Universal Robots URScript: Main Program.script

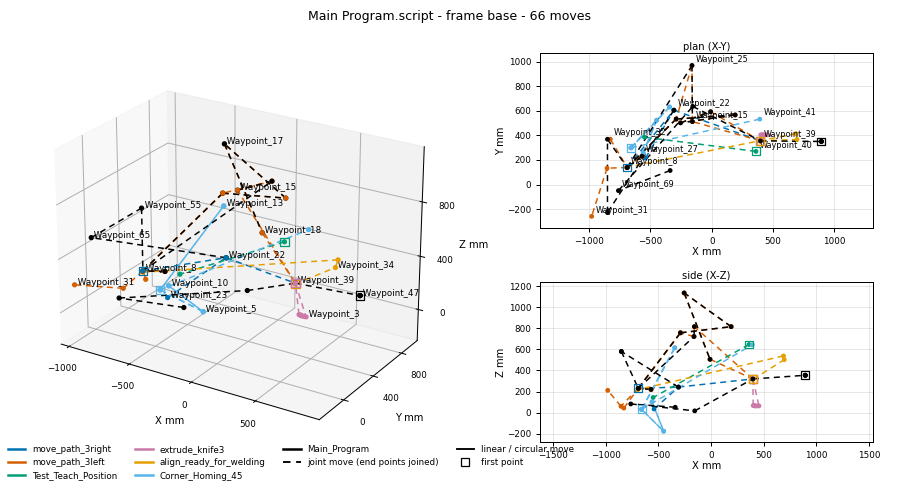
[picture p0: tool path of Main Program.script in frame base, 66 of 133 moves have a stored position in this frame; points joined in program order, loops and branches not executed]
def Main_Program():
  global _hidden_verificationVariable=0
  step_count_c083da12_c088_44e4_86e2_368702bf93a6 = 0.0
  thread Step_Counter_Thread_2b585d60_45ad_46e5_9eb7_fcb77fea0485():
    while (True):
      step_count_c083da12_c088_44e4_86e2_368702bf93a6 = step_count_c083da12_c088_44e4_86e2_368702bf93a6 + 1.0
      sync()
    end
  end
  run Step_Counter_Thread_2b585d60_45ad_46e5_9eb7_fcb77fea0485()
  set_target_payload(10.450000, [0.000000, -0.064000, 0.064000], [0.076889, 0.076889, 0.076889, 0.000000, 0.000000, 0.000000])
  set_tool_communication(False, 115200, 0, 1, 1.5, 3.5)
  set_tool_output_mode(0)
  set_tool_digital_output_mode(0, 1)
  set_tool_digital_output_mode(1, 1)
  set_tool_voltage(0)
  set_safety_mode_transition_hardness(1)
  set_tcp(p[-0.00549,-0.328,0.10639,1.2092,-1.2092,1.2092])
  set_gravity([0.0, 0.0, 9.82])
  set_standard_analog_input_domain(0, 1)
  set_standard_analog_input_domain(1, 1)
  set_tool_analog_input_domain(0, 1)
  set_tool_analog_input_domain(1, 1)
  set_analog_outputdomain(0, 0)
  set_analog_outputdomain(1, 0)
  set_input_actions_to_default()
  global Point_1=p[0.0,0.0,0.0,0.0,0.0,0.0]
  # begin: URCap Installation Node
  #   Source: MachineLogic for Universal Robots, 3.1.7, Vention Inc.
  #   Type: MachineLogic for Universal Robots
  def waitForResponse(expected_response_vention, cname_vention):
  response_vention = socket_read_string(cname_vention,timeout=15)
  while response_vention != expected_response_vention:
  sleep(0.01)
  response_vention = socket_read_string(cname_vention,timeout=15)
  end
  sleep(0.01)
  sync()
  end
  def sendString(string_vention, expected_response_vention, cname_vention):
  socket_send_string(str_cat(string_vention,";"), cname_vention)
  response_vention = socket_read_string(cname_vention,timeout=15)
  if(response_vention == "nAck"):
  popup("nAck received")
  end
  while response_vention != expected_response_vention:
  sleep(0.01)
  response_vention = socket_read_string(cname_vention,timeout=15)
  if(response_vention == "nAck"):
  popup("nAck received")
  end
  end
  sleep(0.01)
  sync()
  end
  def sendStringNAck(string_vention, expected_response_vention, cname_vention):
  socket_send_string(str_cat(string_vention,";"), cname_vention)
  response_vention = socket_read_string(cname_vention,timeout=15)
  if(response_vention == "nAck"):
  popup("nAck received")
  end
  while(response_vention != expected_response_vention and response_vention != "nAck"):
  sleep(0.01)
  response_vention = socket_read_string(cname_vention,timeout=15)
  if(response_vention == "nAck"):
  popup("nAck received",blocking=True)
  end
  end
  sleep(0.01)
  sync()
  end
  def sendStringWithTimeout(string_vention, expected_response_vention, cname_vention):
  socket_send_string(str_cat(string_vention,";"), cname_vention)
  response_vention = socket_read_string(cname_vention,timeout=10)
  if(response_vention == "nAck"):
  popup("nAck received"+string_vention)
  end
  sleep(0.01)
  sync()
  end
  def pollString(string_vention, expected_response_vention, cname_vention):
  socket_send_string(str_cat(string_vention,";"), cname_vention)
  response_vention = socket_read_string(cname_vention,timeout=15)
  if(response_vention == "nAck"):
  popup("nAck received")
  end
  while response_vention != expected_response_vention:
  sleep(1)
  socket_send_string(str_cat(string_vention,";"), cname_vention)
  response_vention = socket_read_string(cname_vention,timeout=15)
  if(response_vention == "nAck"):
  popup("nAck received")
  end
  end
  sleep(0.01)
  sync()
  end
  def sendVariable(var_vention, data_vention, expected_response_vention, cname_vention):
  socket_set_var(var_vention, data_vention, cname_vention)
  response_vention = socket_read_string(cname_vention,timeout=15)
  if(response_vention == "nAck"):
  popup("nAck received")
  end
  while response_vention != expected_response_vention:
  sleep(0.01)
  response_vention = socket_read_string(cname_vention,timeout=15)
  if(response_vention == "nAck"):
  popup("nAck received")
  end
  end
  sleep(0.01)
  sync()
  end
  def intToString(integer_vention,cname_vention):
  stringFix=""
  multiplier_vention123=1
  if integer_vention<0:
  stringFix="-"
  multiplier_vention123=-1
  end
  socket_set_var("GetString",integer_vention*multiplier_vention123,cname_vention)
  string_vention=""
  while string_vention=="":
  sleep(0.01)
  string_vention=socket_read_string(cname_vention,timeout=15)
  end
  sleep(0.01)
  sync()
  string_vention=stringFix+string_vention
  return string_vention
  end
  string_vention=""
  isVentionMovementBusy = False
  isVentionParallelMovementSendingScript = False
  ventionThreadHandle = 1
  isVentionMovementBusyMachineMotion1 = False
  isVentionParallelMovementSendingScriptMachineMotion1 = False
  socket_vention = socket_open("192.168.3.52", 9999, "MachineMotion1")
  if socket_vention==False:
  popup("Check configuration, can't connect to MachineMotion")
  end
  waitForResponse("MachineMotion connection established", "MachineMotion1")
  sendString("isReady", "MachineMotion isReady = true", "MachineMotion1")
  sendStringWithTimeout("setURCapVersion2", "setURCapVersion loaded", "MachineMotion1")
  sendString("SET speed_v2 1000000", "Ack", "MachineMotion1")
  sendString("SET acceleration_v2 100000", "Ack", "MachineMotion1")
  sendString("SET de_axis_1_microsteps_config 8", "Ack", "MachineMotion1")
  sendString("SET de_axis_1_mechanical_gain_config_v2 150000.0", "Ack", "MachineMotion1")
  sendString("SET de_axis_1_direction_config 1", "Ack", "MachineMotion1")
  sendString("SET de_axis_1_type_config Custom Actuator ", "Ack", "MachineMotion1")
  sendString("de_axis_1_config_exec", "Ack", "MachineMotion1")
  # end: URCap Installation Node
  # begin: URCap Installation Node
  #   Source: WireTank Serial, 4.9.0, WireTank, LLC
  #   Type: WireTank Serial
  WTSerialBridge = rpc_factory("xmlrpc","http://127.0.0.1:40511/RPC2")
  # end: URCap Installation Node
  global freedrive_m_var=  False
  global Waypoint_47_p=p[.894110788705, .351078070639, .354441232572, 2.326362155719, 2.052509368646, .057355656444]
  global Waypoint_47_q=[-3.266942326222555, -1.1744836431792756, 1.6532800833331507, 1.0039457517811279, -0.0024531523333948257, -1.5362089315997522]
  global Waypoint_50_p=p[-.568711442653, .230601791901, .220208834751, -1.519093932087, -.535128035721, .573965472012]
  global Waypoint_50_q=[-0.021522347127095998, -1.2794721287539979, 2.4323821703540247, 5.090870934515753, -2.2996109167682093, 1.533644199371338]
  global Waypoint_51_p=p[-.689649894186, .139001107022, .230693120258, -.852023156701, -1.645963115617, 1.645984943001]
  global Waypoint_51_q=[-1.1454814116107386, -1.5427037247321387, 2.8454700152026575, 4.979047852545538, -4.902958456669943, 1.5718834400177002]
  global Waypoint_52_p=p[-.160992057407, .970528182050, .722037363514, -.554955923310, .106486629259, .328544950173]
  global Waypoint_52_q=[-1.2978580633746546, -1.3217003357461472, 2.2583277861224573, 3.7025129038044433, -2.952825371419088, 0.9627944231033325]
  global Waypoint_53_p=p[-.157624488365, .513351401913, .815670293526, -.672704566373, -1.852329693545, -.055423312366]
  global Waypoint_53_q=[-2.7676661650287073, -1.8206430874266566, 2.312763277684347, 1.0122546392628173, -1.0765226523028772, -0.8102834860431116]
  global Waypoint_54_p=p[-.308528116178, .606080777007, .242371251996, -2.133736658076, .349438277129, 2.130953356703]
  global Waypoint_54_q=[-1.9617512861834925, -1.2994225782207032, 2.207935158406393, 0.745708628291748, 1.5955500602722168, 1.41863214969635]
  global Waypoint_65_p=p[-.850299549699, -.229060500451, .580194265918, -.066683564301, -1.566406749139, -.045536147896]
  global Waypoint_65_q=[0.11527767777442932, -1.206728772526123, 2.660132948552267, 3.2525827127644042, -4.69939905801882, -0.18521625200380498]
  global Waypoint_55_p=p[-.850295942693, .369353811615, .580190947871, -.066690142153, -1.566409865149, -.045506050424]
  global Waypoint_55_q=[-0.89636737505068, -1.198587493305542, 2.6061368624316614, 3.3119169908710937, -4.700617257748739, 0.826545238494873]
  global Waypoint_59_p=p[-.689650832419, .138973473550, .230700469426, -.851985360280, -1.645991124348, 1.645990580233]
  global Waypoint_59_q=[-1.1454528013812464, -1.5427289356342335, 2.8454795519458216, 4.979044186859884, -4.902960960065023, 1.5718833208084106]
  global Waypoint_71_p=p[-.289684660393, .534258475721, .757199031184, -.295236718653, -.653013693815, .389426431276]
  global Waypoint_71_q=[-1.3941848913775843, -1.6550847492613734, 2.7336130777942103, 4.156678839320801, -3.798194471989767, 1.7310842275619507]
  global Waypoint_58_p=p[.191120239889, .567518478899, .815512910186, -.135765364935, .396070873472, .208834263225]
  global Waypoint_58_q=[-1.651280705128805, -1.7712346516051234, 2.617981735860006, 3.3066598612019042, -2.656208101903097, 0.8563313484191895]
  global Waypoint_56_p=p[-.254568281661, .502958752129, 1.135400507516, -.261908057482, -.749714619963, 1.349050618455]
  global Waypoint_56_q=[-2.0344861189471644, -1.9012485943236292, 2.469647232686178, 2.2012061315723876, -1.1677187124835413, -0.5094392935382288]
  global Waypoint_57_p=p[-.009221327687, .593713365169, .505808930157, -1.424394189587, -2.344106819810, -.527597949261]
  global Waypoint_57_q=[-2.920837704335348, -1.9932075939574183, 2.3856611887561243, 0.6815890508839111, -0.5688460508929651, -1.1506975332843226]
  global Waypoint_67_p=p[-.339169194335, .114271165560, .051007401747, -.434162127311, 1.872717119498, -1.885153895998]
  global Waypoint_67_q=[-1.410516087208883, -0.9778240484050293, 2.47756010690798, -1.72361483196401, -0.3956816832171839, 1.808600902557373]
  global Waypoint_69_p=p[-.760826542313, -.049762698068, .082649581767, -1.026233921905, -1.612699318499, 1.547123897415]
  global Waypoint_69_q=[-0.22154647508730108, -1.118469015961029, 2.7561236063586634, -1.5568565337783475, -3.851987902318136, 1.559481143951416]
  global Waypoint_70_p=p[-.154414768496, .636923137577, .016979120256, -.302753655748, 1.486961848367, .122240024639]
  global Waypoint_70_q=[-1.1281922499286097, -1.0678585332683106, 2.4290812651263636, -2.7994214497008265, -1.6034835020648401, 1.7401196956634521]
  global Waypoint_49_p=p[.397354147848, .356263001249, .319808682466, 2.316306590727, 2.057646408591, .074101958728]
  global Waypoint_49_q=[-3.4579480330096644, -2.0568953953185023, 2.3266006151782435, -0.2270372670939942, -0.1993797461139124, -0.10534602800478154]
  global Waypoint_48_p=p[.894089819959, .351089510856, .354452935433, 2.326359030986, 2.052526986878, .057346871716]
  global Waypoint_48_q=[-3.266932551060812, -1.1745034915259858, 1.653294865285055, 1.0039614874073486, -0.002454582844869435, -1.5362089315997522]
  global Waypoint_46_p=p[.894107867742, .351078231601, .354456446052, 2.326366960603, 2.052510258679, .057358671808]
  global Waypoint_46_q=[-3.266944233571188, -1.1744955343059083, 1.6532734076129358, 1.003952904338501, -0.002457443867818654, -1.5361955801593226]
  global Waypoint_8_p=p[-.689650873132, .138963273545, .230691387978, -.851994598965, -1.645998530536, 1.646007616333]
  global Waypoint_8_q=[-0.9414032141314905, -1.501500443821289, 2.801856819783346, 4.981602895050802, -4.698942009602682, 1.571649193763733]
  global Waypoint_22_p=p[-.308534453517, .606084664264, .242393158856, 1.369873371142, 1.066881263643, -1.257197506198]
  global Waypoint_22_q=[-1.4685500303851526, -0.9664557737163086, 1.6195090452777308, 0.9282776552387695, 1.6574476957321167, 0.2630845010280609]
  global Waypoint_23_p=p[-.540166575654, .215949141041, .034631452617, -1.505795438113, 1.057579835594, 1.573514753692]
  global Waypoint_23_q=[-0.46167117754091436, -1.1365486842444916, 2.508885685597555, 0.15223841249432368, 1.4952874183654785, 3.819530963897705]
  global Waypoint_24_p=p[-.308525559537, .606096497354, .242373144855, -2.133742737559, .349425192770, 2.130939839044]
  global Waypoint_24_q=[-1.8709262053119105, -1.2877716285041352, 2.192875687276022, 0.7510036665150146, 1.5878156423568726, 1.5091480016708374]
  global Waypoint_39_p=p[.397377312153, .356253310648, .319810281486, 2.316317670744, 2.057592854035, .074120023159]
  global Waypoint_39_q=[-3.4579551855670374, -2.0568958721556605, 2.3265963236438196, -0.22706706941638188, -0.19935590425600225, -0.10534030595888311]
  global Waypoint_37_p=p[.397366630181, .356258644196, .319813668943, 2.316299214281, 2.057614642521, .074125657910]
  global Waypoint_37_q=[-3.4579508940326136, -2.056904455224508, 2.3265963236438196, -0.2270481151393433, -0.19937020937074834, -0.10535222688783819]
  global Waypoint_15_p=p[-.157621040248, .513353603496, .815677694745, -.672699538592, -1.852318447516, -.055422773001]
  global Waypoint_15_q=[-2.770456854497091, -1.8207680187621058, 2.3065691629992884, 1.0170823770710449, -1.0767205397235315, -0.8071182409869593]
  global Waypoint_25_p=p[-.161036555831, .970524399959, .722042384791, -.554954311189, .106465018540, .328580879483]
  global Waypoint_25_q=[-1.3071630636798304, -1.3366777312806626, 2.2083633581744593, 3.7187773424335937, -2.9519384543048304, 0.9132363796234131]
  global Waypoint_72_p=p[-.289685725237, .534256396594, .757196155975, -.295237726329, -.653009715205, .389435972469]
  global Waypoint_72_q=[-1.394179646168844, -1.6550847492613734, 2.7336154619800013, 4.156686468715332, -3.7981911341296595, 1.731092095375061]
  global Waypoint_26_p=p[-.689650873132, .138963273545, .230691387978, -.851994598965, -1.645998530536, 1.646007616333]
  global Waypoint_26_q=[-0.9414032141314905, -1.501500443821289, 2.801856819783346, 4.981602895050802, -4.698942009602682, 1.571649193763733]
  global Waypoint_27_p=p[-.568724745609, .230601805298, .220208295176, -1.519097711196, -.535155391172, .573964121010]
  global Waypoint_27_q=[-0.04883271852602178, -1.2753942471793671, 2.4771457354175013, 5.041022258787908, -2.326899592076437, 1.532160997390747]
  global Waypoint_28_p=p[-.568724745609, .230601805298, .220208295176, -1.519097711196, -.535155391172, .573964121010]
  global Waypoint_28_q=[-0.04883271852602178, -1.2753942471793671, 2.4771457354175013, 5.041022258787908, -2.326899592076437, 1.532160997390747]
  global Waypoint_29_p=p[-.689650873132, .138963273545, .230691387978, -.851994598965, -1.645998530536, 1.646007616333]
  global Waypoint_29_q=[-0.9414032141314905, -1.501500443821289, 2.801856819783346, 4.981602895050802, -4.698942009602682, 1.571649193763733]
  global Waypoint_30_p=p[-.853851193668, .133266829906, .060418082908, -.274178222953, -2.359710051999, .046821166283]
  global Waypoint_30_q=[-0.608560864125387, -1.0122360748103638, 2.787060801182882, 3.7283646303364257, -4.940747324620382, 0.3777344226837158]
  global Waypoint_31_p=p[-.979398188272, -.259625449453, .211289397035, -.673010443572, -1.459355862765, -.640164958946]
  global Waypoint_31_q=[0.36968713998794556, -0.5732358259013672, 2.138303581868307, 3.1253925996967773, -4.70385724702944, -1.2100523153888147]
  global Waypoint_32_p=p[-.826865752305, .369357632284, .043113676955, .574997346548, -1.492225541214, .597128135378]
  global Waypoint_32_q=[-1.0355513731585901, -0.33930082738909917, 2.126244846974508, 2.9386045175739746, -4.711197797452108, 1.7860286235809326]
  global Waypoint_33_p=p[-.689650873132, .138963273545, .230691387978, -.851994598965, -1.645998530536, 1.646007616333]
  global Waypoint_33_q=[-0.9414032141314905, -1.501500443821289, 2.801856819783346, 4.981602895050802, -4.698942009602682, 1.571649193763733]
  global Waypoint_73_p=p[-.289671192632, .534275423553, .757232902417, -.295189983811, -.652980753171, .389398176275]
  global Waypoint_73_q=[-1.39418870607485, -1.65509094814443, 2.7335642019854944, 4.156684561366699, -3.7981610933886927, 1.731088399887085]
  global Waypoint_16_p=p[.191112811238, .567512170908, .815514010937, -.135771161622, .396053809900, .208825693369]
  global Waypoint_16_q=[-1.6536315123187464, -1.762029310266012, 2.6225650946246546, 3.2891055780598144, -2.6549678484546106, 0.8520665764808655]
  global Waypoint_17_p=p[-.254565633623, .502963426820, 1.135401557820, -.261910507478, -.749716086887, 1.349041636154]
  global Waypoint_17_q=[-2.035229508076803, -1.8928028545775355, 2.468372408543722, 2.19391576826062, -1.167032543812887, -0.5091407934771937]
  global Waypoint_18_p=p[-.009208376822, .593717720951, .505810027228, -1.424406033077, -2.344120510145, -.527630245278]
  global Waypoint_18_q=[-2.9172328154193323, -1.9945279560484828, 2.3804522196399134, 0.6930715280720214, -0.5671199003802698, -1.1566088835345667]
  global Waypoint_38_p=p[.397379749540, .356252016937, .319817140705, 2.316310534508, 2.057580214841, .074134378577]
  global Waypoint_38_q=[-3.457958761845724, -2.0569073162474574, 2.3265913168536585, -0.22705944002185063, -0.19935638109316045, -0.10534793535341436]
  global Waypoint_40_p=p[.360688403366, .270119715397, .646144746546, .057805349154, 2.125995180379, 2.134053153683]
  global Waypoint_40_q=[-3.4579489866839808, -2.0569035015501917, 2.3265796343432825, -0.22706706941638188, -0.1993501822101038, -0.10534793535341436]
  global Waypoint_2_p=p[-.548957282596, .386284559177, .143710178207, 1.570800598292, -.000025190822, .000004803470]
  global Waypoint_2_q=[-1.0516188780414026, -1.010990933781006, 2.1562450567828577, -1.143702046280243, -1.0526168982135218, -0.0017235914813440445]
  global Waypoint_20_p=p[.397380247322, .356253634699, .319820846021, 2.316316320871, 2.057594704604, .074118471609]
  global Waypoint_20_q=[-3.457949940358297, -2.056894441644186, 2.32658034959902, -0.2270551484874268, -0.19935208955873662, -0.10533696809877569]
  global Waypoint_3_p=p[.454852104155, .405448828659, .064015413765, 2.316807606413, 2.051392071696, .076664825947]
  global Waypoint_3_q=[-3.274653975163595, -1.5604325172356148, 2.467809502278463, -0.34438879907641606, -0.014281574879781544, -0.6303489843951624]
  global Waypoint_21_p=p[.439068323950, .405460163829, .064006334409, 2.316810979609, 2.051438029044, .076624763552]
  global Waypoint_21_q=[-3.2805374304400843, -1.6257621250548304, 2.5041499773608606, -0.4786943954280396, -0.019728008900777638, -0.46699268022646123]
  global Waypoint_42_p=p[.421302935105, .405445303018, .063010865956, 2.316845912097, 2.051376323407, .076625998808]
  global Waypoint_42_q=[-3.2879136244403284, -1.6787048778929652, 2.5389068762408655, -0.5691380065730591, -0.02675801912416631, -0.35834962526430303]
  global Waypoint_43_p=p[.417011768852, .405435328663, .065002627117, 2.316867113472, 2.051334925313, .076628493429]
  global Waypoint_43_q=[-3.289830032979147, -1.6934038601317347, 2.5445857683764856, -0.579618052845337, -0.028589550648824513, -0.33885270753969365]
  global Waypoint_44_p=p[.413030241071, .405436708516, .067007287168, 2.316842962602, 2.051343797062, .076642826315]
  global Waypoint_44_q=[-3.291628662739889, -1.7069231472411097, 2.5494325796710413, -0.5873385828784485, -0.03035623231996709, -0.3224685827838343]
  global Waypoint_74_p=p[.400006724768, .405435114685, .067002832650, 2.316857393772, 2.051322715522, .076640196251]
  global Waypoint_74_q=[-3.2978647390948694, -1.7389985523619593, 2.5696502367602747, -0.6192590159228821, -0.03645164171327764, -0.27867013612856084]
  global Waypoint_45_p=p[.397380247322, .356253634699, .319820846021, 2.316316320871, 2.057594704604, .074118471609]
  global Waypoint_45_q=[-3.457949940358297, -2.056894441644186, 2.32658034959902, -0.2270551484874268, -0.19935208955873662, -0.10533696809877569]
  global oldhome_p=p[.397683836105, .356251384911, .315246899233, 2.316304177919, 2.057561756051, .074146544723]
  global oldhome_q=[-3.457960907612936, -2.0569125614561976, 2.326589886342184, -0.22707636774096684, -0.19935208955873662, -0.10534269014467412]
  global Waypoint_34_p=p[.695155464390, .367451880816, .502522491683, 2.093108370749, 1.857548644474, .308841595089]
  global Waypoint_34_q=[-3.249415699635641, -1.9387923679747523, 2.3226097265826624, 3.981850786800049, -0.05697328249086553, 1.5286790132522583]
  global Waypoint_35_p=p[.687527620967, .415165960724, .537921070000, 2.127101811831, 1.929915403723, .470130777221]
  global Waypoint_35_q=[-3.249424997960226, -1.9387947521605433, 2.32263428369631, 3.9818588930317382, -6.198007937763826, 1.5286580324172974]
  global Waypoint_36_p=p[-.693756081485, .141369193308, .218584735520, -.851978179689, -1.646001533937, 1.646008371360]
  global Waypoint_36_q=[-1.1533568541156214, -1.4924076360515137, 2.8518698851214808, 4.922323781042852, -4.910887185727255, 1.5719373226165771]
  def calculate_point_to_move_towards(feature, direction, position_distance):
    local posDir=[direction[0], direction[1], direction[2]]
    if (norm(posDir) < 1e-6):
      return get_target_waypoint()
    end
    local direction_vector_normalized=normalize(posDir)
    local displacement_pose=p[direction_vector_normalized[0] * position_distance,direction_vector_normalized[1] * position_distance,direction_vector_normalized[2] * position_distance,0,0,0]
    local wanted_displacement_in_base_frame=pose_sub(pose_trans(feature, displacement_pose), feature)
    return pose_add(get_target_waypoint(), wanted_displacement_in_base_frame)
  end
  global Waypoint_4_p=p[-.658264763546, .299530128456, .030909835036, .426821001551, -1.621505068649, .437070885767]
  global Waypoint_4_q=[-1.350241486226217, -0.9702387017062684, 2.492185179387228, -1.7834822140135707, -0.33723670641054326, 1.8489984273910522]
  global Waypoint_5_p=p[-.448862677341, .524599667441, -.175967040878, 2.473330473302, -1.874382924863, .205319206046]
  global Waypoint_5_q=[-1.1354392210589808, -1.0039964479259034, 2.441021744404928, -2.875528474847311, -1.6043828169452112, 1.7329596281051636]
  global Waypoint_10_p=p[-.559130451394, .259233925829, .102445980692, -.822649281727, -1.486064670292, -.881476138414]
  global Waypoint_10_q=[-0.556256119404928, -1.0744255942157288, 2.9114087263690394, -1.7763501606383265, -4.185837809239523, 1.5288889408111572]
  global Waypoint_11_p=p[-.559130451394, .259233925829, .102445980692, -.822649281727, -1.486064670292, -.881476138414]
  global Waypoint_11_q=[-0.556256119404928, -1.0744255942157288, 2.9114087263690394, -1.7763501606383265, -4.185837809239523, 1.5288889408111572]
  global Waypoint_12_p=p[-.448862677341, .524599667441, -.175967040878, 2.473330473302, -1.874382924863, .205319206046]
  global Waypoint_12_q=[-1.1354392210589808, -1.0039964479259034, 2.441021744404928, -2.875528474847311, -1.6043828169452112, 1.7329596281051636]
  global Waypoint_13_p=p[-.343952006273, .632142227752, .615174722549, -.025948978133, -.008794819136, -.567469912202]
  global Waypoint_13_q=[-1.350241486226217, -0.9702451390079041, 2.492171827946798, -3.0669099293150843, 1.575993537902832, 2.355180025100708]
  global Waypoint_14_p=p[-.343952006273, .632142227752, .615174722549, -.025948978133, -.008794819136, -.567469912202]
  global Waypoint_14_q=[-1.350241486226217, -0.9702451390079041, 2.492171827946798, -3.0669099293150843, 1.575993537902832, 2.355180025100708]
  global Waypoint_41_p=p[.392127936214, .533269017847, .644148583936, .057822570580, 2.125982462550, 2.134033989912]
  global Waypoint_41_q=[-3.4579578081714075, -2.0569120846190394, 2.3265841642962855, -0.22706885755572515, -0.1993349234210413, -0.10534984270204717]
  def move_path_3right():
    $ 118 "move_path_3right" "noBreak"
    $ 119 "'this is the path for Down, Over, then Back Around'"
    # 'this is the path for Down, Over, then Back Around'
    $ 120 "Comment"
    # Comment
    $ 129 "align_ready_for_welding()"
    align_ready_for_welding()
    $ 130 "Comment"
    # Comment
    $ 131 "p1≔pathturn[0]"
    global p1=pathturn[0]
    $ 132 "p2≔pathturn[1]"
    global p2=pathturn[1]
    $ 133 "p4≔pathturn[2]"
    global p4=pathturn[2]
    $ 134 "p5≔pathturn[3]"
    global p5=pathturn[3]
    $ 135 "MoveJ"
    $ 136 "p1" "breakAfter"
    movej(p1, a=1.3962634015954636, v=1.0471975511965976)
    $ 137 "Wait: 8.0"
    sleep(8.0)
    $ 140 "turn_extrusion_on()"
    turn_extrusion_on()
    $ 141 "Set DO[0]=On"
    set_standard_digital_out(0, True)
    $ 142 "MoveL"
    $ 143 "p2" "breakAfter"
    movel(p2, a=0.1, v=0.01)
    # begin: URCap Program Node
    #   Source: WireTank Serial, 4.9.0, WireTank, LLC
    #   Type: WireTank Serial
    $ 144 "Serial Bridge uR0"
    SerialResponse = WTSerialBridge.send_command("/dev/ttyUSB0",1200, 8, "None", "One", "None", 1000, "None", "None", [252,82,48], False)
    # end: URCap Program Node
    $ 145 "Wait: 0.5"
    sleep(0.5)
    $ 146 "Set DO[0]=Off"
    set_standard_digital_out(0, False)
    $ 147 "MoveL"
    $ 148 "p4" "breakAfter"
    movel(p4, a=0.01, v=0.12)
    $ 151 "turn_extrusion_on()"
    turn_extrusion_on()
    $ 152 "Set DO[0]=On"
    set_standard_digital_out(0, True)
    $ 153 "MoveL"
    $ 154 "p5" "breakAfter"
    movel(p5, a=0.1, v=0.01)
    # begin: URCap Program Node
    #   Source: WireTank Serial, 4.9.0, WireTank, LLC
    #   Type: WireTank Serial
    $ 155 "Serial Bridge uR0"
    SerialResponse = WTSerialBridge.send_command("/dev/ttyUSB0",1200, 8, "None", "One", "None", 1000, "None", "None", [252,82,48], False)
    # end: URCap Program Node
    $ 156 "Wait: 2.0"
    sleep(2.0)
    $ 157 "Set DO[0]=Off"
    set_standard_digital_out(0, False)
    $ 158 "Comment"
    # Comment
    $ 159 "pret1≔p[p5[0]+.1,p5[1],p5[2],p5[3],p5[4],p5[5]]"
    global pret1=p[p5[0]+.1,p5[1],p5[2],p5[3],p5[4],p5[5]]
    $ 160 "p_1≔pathturn[4]"
    global p_1=pathturn[4]
    $ 161 "p_2≔pathturn[5]"
    global p_2=pathturn[5]
    $ 162 "p_3≔pathturn[6]"
    global p_3=pathturn[6]
    $ 163 "p_4≔pathturn[7]"
    global p_4=pathturn[7]
    $ 164 "p_5≔pathturn[8]"
    global p_5=pathturn[8]
    $ 165 "p_preheat≔p[p_3[0]+.01,p_3[1],p_3[2],p_3[3],p_3[4],p_3[5]]"
    global p_preheat=p[p_3[0]+.01,p_3[1],p_3[2],p_3[3],p_3[4],p_3[5]]
    $ 166 "p_pre_ret≔p[p_1[0]+.03,p_1[1]+.03,p_1[2],p_1[3],p_1[4],p_1[5]]"
    global p_pre_ret=p[p_1[0]+.03,p_1[1]+.03,p_1[2],p_1[3],p_1[4],p_1[5]]
    $ 167 "p_pre_ret2≔p[p_3[0]+.1,p_3[1],p_3[2],p_3[3],p_3[4],p_3[5]]"
    global p_pre_ret2=p[p_3[0]+.1,p_3[1],p_3[2],p_3[3],p_3[4],p_3[5]]
    $ 168 "MoveJ"
    $ 169 "pret1" "breakAfter"
    movej(pret1, a=1.3962634015954636, v=1.3962634015954636)
    $ 170 "Waypoint_8" "breakAfter"
    movej(get_inverse_kin(Waypoint_8_p, qnear=Waypoint_8_q), a=1.3962634015954636, v=1.0471975511965976)
    $ 172 "Waypoint_22" "breakAfter"
    movej(get_inverse_kin(Waypoint_22_p, qnear=Waypoint_22_q), a=1.3962634015954636, v=1.3962634015954636)
    $ 173 "'preheat'"
    # 'preheat'
    $ 174 "MoveJ"
    $ 175 "p_pre_ret" "breakAfter"
    movej(p_pre_ret, a=1.3962634015954636, v=1.0471975511965976)
    $ 176 "p_pre_ret2" "breakAfter"
    movej(p_pre_ret2, a=1.3962634015954636, v=1.0471975511965976)
    $ 177 "p_preheat" "breakAfter"
    movej(p_preheat, a=1.3962634015954636, v=1.0471975511965976)
    $ 178 "Wait: 8.0"
    sleep(8.0)
    $ 179 "MoveJ"
    $ 180 "p_pre_ret2" "breakAfter"
    movej(p_pre_ret2, a=1.3962634015954636, v=1.0471975511965976)
    $ 181 "p_pre_ret" "breakAfter"
    movej(p_pre_ret, a=1.3962634015954636, v=1.0471975511965976)
    $ 182 "Set"
    set_tcp(p[0.00451,-0.328,0.10639,1.2092,-1.2092,1.2092])
    $ 183 "MoveL"
    $ 184 "p_1" "breakAfter"
    movel(p_1, a=1.2, v=0.05)
    $ 187 "Set DO[0]=On"
    set_standard_digital_out(0, True)
    $ 188 "turn_extrusion_on()"
    turn_extrusion_on()
    $ 189 "MoveL"
    $ 190 "p_2" "breakAfter"
    movel(p_2, a=1.2, v=0.02)
    $ 191 "MoveP"
    $ 192 "CircleMove"
    $ 193 "p_3" "noBreak"
    $ 194 "p_4" "breakAfter"
    movec(p_3, p_4, a=0.01, v=0.001, r=0.0, mode=1)
    $ 195 "MoveL"
    $ 196 "p_5" "breakAfter"
    movel(p_5, a=1.2, v=0.012)
    # begin: URCap Program Node
    #   Source: WireTank Serial, 4.9.0, WireTank, LLC
    #   Type: WireTank Serial
    $ 197 "Serial Bridge uR0"
    SerialResponse = WTSerialBridge.send_command("/dev/ttyUSB0",1200, 8, "None", "One", "None", 1000, "None", "None", [252,82,48], False)
    # end: URCap Program Node
    $ 198 "Wait: 2.0"
    sleep(2.0)
    $ 199 "Set DO[0]=Off"
    set_standard_digital_out(0, False)
    $ 200 "MoveL"
    $ 201 "Waypoint_23" "breakAfter"
    movel(Waypoint_23_p, a=1.2, v=0.25)
    $ 202 "MoveJ"
    $ 203 "Waypoint_24" "breakAfter"
    movej(get_inverse_kin(Waypoint_24_p, qnear=Waypoint_24_q), a=1.3962634015954636, v=1.0471975511965976)
    $ 204 "Waypoint_39" "breakAfter"
    movej(get_inverse_kin(Waypoint_39_p, qnear=Waypoint_39_q), a=1.3962634015954636, v=1.0471975511965976)
    $ 205 "'above waypoint is home'"
    # 'above waypoint is home'
  end
  def move_path_3left():
    $ 206 "move_path_3left" "noBreak"
    $ 207 "'this is the path for Down, Over, then Back Around'"
    # 'this is the path for Down, Over, then Back Around'
    $ 208 "Comment"
    # Comment
    $ 209 "MoveJ"
    $ 210 "Waypoint_37" "breakAfter"
    movej(get_inverse_kin(Waypoint_37_p, qnear=Waypoint_37_q), a=1.3962634015954636, v=1.0471975511965976)
    $ 211 "'above point is home'"
    # 'above point is home'
    $ 212 "Waypoint_15" "breakAfter"
    movej(get_inverse_kin(Waypoint_15_p, qnear=Waypoint_15_q), a=1.3962634015954636, v=1.0471975511965976)
    $ 213 "Waypoint_25" "breakAfter"
    movej(get_inverse_kin(Waypoint_25_p, qnear=Waypoint_25_q), a=1.3962634015954636, v=1.0471975511965976)
    $ 214 "Waypoint_72" "breakAfter"
    movej(get_inverse_kin(Waypoint_72_p, qnear=Waypoint_72_q), a=1.3962634015954636, v=1.0471975511965976)
    $ 215 "Waypoint_26" "breakAfter"
    movej(get_inverse_kin(Waypoint_26_p, qnear=Waypoint_26_q), a=1.3962634015954636, v=1.0471975511965976)
    $ 216 "Waypoint_27" "breakAfter"
    movej(get_inverse_kin(Waypoint_27_p, qnear=Waypoint_27_q), a=1.3962634015954636, v=1.0471975511965976)
    $ 221 "Comment"
    # Comment
    $ 222 "p1≔pathturn[0]"
    global p1=pathturn[0]
    $ 223 "p2≔pathturn[1]"
    global p2=pathturn[1]
    $ 224 "p4≔pathturn[2]"
    global p4=pathturn[2]
    $ 225 "p5≔pathturn[3]"
    global p5=pathturn[3]
    $ 226 "pa1≔p[p1[0]+0.05,p1[1]-0.05,p1[2],p1[3],p1[4],p1[5]]"
    global pa1=p[p1[0]+0.05,p1[1]-0.05,p1[2],p1[3],p1[4],p1[5]]
    $ 227 "MoveJ"
    $ 228 "pa1" "breakAfter"
    movej(pa1, a=1.3962634015954636, v=1.0471975511965976)
    $ 229 "MoveJ"
    $ 230 "p1" "breakAfter"
    movej(p1, a=1.3962634015954636, v=0.2617993877991494)
    $ 231 "Wait: 8.0"
    sleep(8.0)
    $ 234 "turn_extrusion_on()"
    turn_extrusion_on()
    $ 235 "Set DO[0]=On"
    set_standard_digital_out(0, True)
    $ 236 "MoveL"
    $ 237 "p2" "breakAfter"
    movel(p2, a=0.1, v=0.01)
    # begin: URCap Program Node
    #   Source: WireTank Serial, 4.9.0, WireTank, LLC
    #   Type: WireTank Serial
    $ 238 "Serial Bridge uR0"
    SerialResponse = WTSerialBridge.send_command("/dev/ttyUSB0",1200, 8, "None", "One", "None", 1000, "None", "None", [252,82,48], False)
    # end: URCap Program Node
    $ 239 "Wait: 0.5"
    sleep(0.5)
    $ 240 "Set DO[0]=Off"
    set_standard_digital_out(0, False)
    $ 241 "MoveL"
    $ 242 "p4" "breakAfter"
    movel(p4, a=0.01, v=0.12)
    $ 245 "turn_extrusion_on()"
    turn_extrusion_on()
    $ 246 "Set DO[0]=On"
    set_standard_digital_out(0, True)
    $ 247 "MoveL"
    $ 248 "p5" "breakAfter"
    movel(p5, a=0.1, v=0.01)
    # begin: URCap Program Node
    #   Source: WireTank Serial, 4.9.0, WireTank, LLC
    #   Type: WireTank Serial
    $ 249 "Serial Bridge uR0"
    SerialResponse = WTSerialBridge.send_command("/dev/ttyUSB0",1200, 8, "None", "One", "None", 1000, "None", "None", [252,82,48], False)
    # end: URCap Program Node
    $ 250 "Wait: 2.0"
    sleep(2.0)
    $ 251 "Set DO[0]=Off"
    set_standard_digital_out(0, False)
    $ 252 "Comment"
    # Comment
    $ 253 "pret1≔p[p5[0]+.1,p5[1],p5[2],p5[3],p5[4],p5[5]]"
    global pret1=p[p5[0]+.1,p5[1],p5[2],p5[3],p5[4],p5[5]]
    $ 254 "p_1≔pathturn[4]"
    global p_1=pathturn[4]
    $ 255 "p_2≔pathturn[5]"
    global p_2=pathturn[5]
    $ 256 "p_3≔pathturn[6]"
    global p_3=pathturn[6]
    $ 257 "p_4≔pathturn[7]"
    global p_4=pathturn[7]
    $ 258 "p_5≔pathturn[8]"
    global p_5=pathturn[8]
    $ 259 "p_preheat≔p[p_3[0]+.01,p_3[1],p_3[2],p_3[3],p_3[4],p_3[5]]"
    global p_preheat=p[p_3[0]+.01,p_3[1],p_3[2],p_3[3],p_3[4],p_3[5]]
    $ 260 "p_pre_ret≔p[p_1[0]+.03,p_1[1]-.03,p_1[2],p_1[3],p_1[4],p_1[5]]"
    global p_pre_ret=p[p_1[0]+.03,p_1[1]-.03,p_1[2],p_1[3],p_1[4],p_1[5]]
    $ 261 "p_pre_ret2≔p[p_3[0]+.03,p_3[1],p_3[2],p_3[3],p_3[4],p_3[5]]"
    global p_pre_ret2=p[p_3[0]+.03,p_3[1],p_3[2],p_3[3],p_3[4],p_3[5]]
    $ 262 "MoveJ"
    $ 263 "pret1" "breakAfter"
    movej(pret1, a=1.3962634015954636, v=1.3962634015954636)
    $ 264 "Waypoint_28" "breakAfter"
    movej(get_inverse_kin(Waypoint_28_p, qnear=Waypoint_28_q), a=1.3962634015954636, v=1.3962634015954636)
    $ 265 "'now go into the ccw weld position'"
    # 'now go into the ccw weld position'
    $ 266 "Waypoint_29" "breakAfter"
    movej(get_inverse_kin(Waypoint_29_p, qnear=Waypoint_29_q), a=1.3962634015954636, v=1.3962634015954636)
    $ 267 "Comment"
    # Comment
    $ 268 "Waypoint_30" "breakAfter"
    movej(get_inverse_kin(Waypoint_30_p, qnear=Waypoint_30_q), a=1.3962634015954636, v=1.3962634015954636)
    $ 269 "Waypoint_31" "breakAfter"
    movej(get_inverse_kin(Waypoint_31_p, qnear=Waypoint_31_q), a=1.3962634015954636, v=1.3962634015954636)
    $ 278 "MoveL"
    $ 279 "p_pre_ret" "breakAfter"
    movel(p_pre_ret, a=1.2, v=0.25)
    $ 280 "p_pre_ret2" "breakAfter"
    movel(p_pre_ret2, a=1.2, v=0.25)
    $ 281 "p_preheat" "breakAfter"
    movel(p_preheat, a=1.2, v=0.25)
    $ 282 "Wait: 8.0"
    sleep(8.0)
    $ 283 "MoveL"
    $ 284 "p_pre_ret2" "breakAfter"
    movel(p_pre_ret2, a=1.2, v=0.25)
    $ 285 "p_pre_ret" "breakAfter"
    movel(p_pre_ret, a=1.2, v=0.25)
    $ 286 "Set"
    set_tcp(p[0.00451,-0.328,0.10639,1.2092,-1.2092,1.2092])
    $ 287 "MoveL"
    $ 288 "p_1" "breakAfter"
    movel(p_1, a=1.2, v=0.05)
    $ 291 "Set DO[0]=On"
    set_standard_digital_out(0, True)
    $ 292 "turn_extrusion_on()"
    turn_extrusion_on()
    $ 293 "MoveL"
    $ 294 "p_2" "breakAfter"
    movel(p_2, a=1.2, v=0.02)
    $ 295 "MoveP"
    $ 296 "CircleMove"
    $ 297 "p_3" "noBreak"
    $ 298 "p_4" "breakAfter"
    movec(p_3, p_4, a=0.01, v=0.001, r=0.0, mode=1)
    $ 299 "MoveL"
    $ 300 "p_5" "breakAfter"
    movel(p_5, a=1.2, v=0.012)
    # begin: URCap Program Node
    #   Source: WireTank Serial, 4.9.0, WireTank, LLC
    #   Type: WireTank Serial
    $ 301 "Serial Bridge uR0"
    SerialResponse = WTSerialBridge.send_command("/dev/ttyUSB0",1200, 8, "None", "One", "None", 1000, "None", "None", [252,82,48], False)
    # end: URCap Program Node
    $ 302 "Wait: 2.0"
    sleep(2.0)
    $ 303 "Set DO[0]=Off"
    set_standard_digital_out(0, False)
    $ 308 "MoveJ"
    $ 309 "Waypoint_32" "breakAfter"
    movej(get_inverse_kin(Waypoint_32_p, qnear=Waypoint_32_q), a=1.3962634015954636, v=1.0471975511965976)
    $ 310 "Waypoint_33" "breakAfter"
    movej(get_inverse_kin(Waypoint_33_p, qnear=Waypoint_33_q), a=1.3962634015954636, v=1.0471975511965976)
    $ 311 "Waypoint_73" "breakAfter"
    movej(get_inverse_kin(Waypoint_73_p, qnear=Waypoint_73_q), a=1.3962634015954636, v=1.0471975511965976)
    $ 312 "Comment"
    # Comment
    $ 313 "MoveJ"
    $ 314 "Waypoint_16" "breakAfter"
    movej(get_inverse_kin(Waypoint_16_p, qnear=Waypoint_16_q), a=1.3962634015954636, v=1.0471975511965976)
    $ 315 "Waypoint_17" "breakAfter"
    movej(get_inverse_kin(Waypoint_17_p, qnear=Waypoint_17_q), a=1.3962634015954636, v=1.0471975511965976)
    $ 316 "Waypoint_18" "breakAfter"
    movej(get_inverse_kin(Waypoint_18_p, qnear=Waypoint_18_q), a=1.3962634015954636, v=1.0471975511965976)
    $ 317 "Waypoint_38" "breakAfter"
    movej(get_inverse_kin(Waypoint_38_p, qnear=Waypoint_38_q), a=1.3962634015954636, v=1.0471975511965976)
    $ 318 "'above point is home'"
    # 'above point is home'
  end
  def Test_Teach_Position():
    $ 319 "Test_Teach_Position" "noBreak"
    $ 323 "MoveJ"
    $ 324 "Waypoint_40" "breakAfter"
    set_tcp(p[0.0,0.0,0.019,0.0,0.0,0.0])
    movej(get_inverse_kin(Waypoint_40_p, qnear=Waypoint_40_q), a=1.3962634015954636, v=1.0471975511965976)
    $ 325 "'above waypoint is home'"
    # 'above waypoint is home'
    $ 326 "Waypoint_2" "breakAfter"
    set_tcp(p[0.0,0.0,0.019,0.0,0.0,0.0])
    movej(get_inverse_kin(Waypoint_2_p, qnear=Waypoint_2_q), a=1.3962634015954636, v=1.0471975511965976)
    $ 327 "freedrive_m_var≔ False "
    global freedrive_m_var=  False
    $ 328 "freedrive_m_var≔ True "
    global freedrive_m_var=  True
    $ 329 "Popup: Move the robot to the peg center, then click 'Continue'"
    popup("Move the robot to the peg center, then click 'Continue'", "Message", False, False, blocking=True)
    $ 330 "freedrive_m_var≔ False "
    global freedrive_m_var=  False
    $ 331 "Wait: 0.25"
    sleep(0.25)
    $ 332 "sync()"
    sync()
    $ 333 "tcp_pose≔get_actual_joint_positions()"
    global tcp_pose= get_actual_joint_positions ()
  end
  def align_tcp_left():
    $ 334 "align_tcp_left" "noBreak"
    $ 335 "'this program aligns the tcp parallel to the y direction'"
    # 'this program aligns the tcp parallel to the y direction'
    $ 336 "cp≔get_actual_tcp_pose()"
    global cp= get_actual_tcp_pose ()
    $ 337 "aligned_y_pose≔p[cp[0],cp[1],cp[2],1.570796,0,0]"
    global aligned_y_pose=p[cp[0],cp[1],cp[2],1.570796,0,0]
    $ 338 "MoveJ"
    $ 339 "aligned_y_pose" "breakAfter"
    movej(aligned_y_pose, a=1.3962634015954636, v=1.0471975511965976)
  end
  def extrude_knife3():
    $ 340 "extrude_knife3" "noBreak"
    $ 342 "Set"
    set_tcp(p[-0.00549,-0.328,0.10639,1.2092,-1.2092,1.2092])
    $ 343 "MoveJ"
    $ 344 "Waypoint_20" "breakAfter"
    movej(get_inverse_kin(Waypoint_20_p, qnear=Waypoint_20_q), a=1.3962634015954636, v=1.0471975511965976)
    $ 345 "'above waypoint is home'"
    # 'above waypoint is home'
    $ 346 "'move above bucket'"
    # 'move above bucket'
    $ 347 "MoveJ"
    $ 348 "Waypoint_3" "breakAfter"
    movej(get_inverse_kin(Waypoint_3_p, qnear=Waypoint_3_q), a=1.3962634015954636, v=1.0471975511965976)
    $ 349 "'extrude out a foot'"
    # 'extrude out a foot'
    $ 351 "Set DO[0]=On"
    set_standard_digital_out(0, True)
    $ 352 "turn_extrusion_on()"
    turn_extrusion_on()
    $ 353 "Wait: 24.0"
    sleep(24.0)
    # begin: URCap Program Node
    #   Source: WireTank Serial, 4.9.0, WireTank, LLC
    #   Type: WireTank Serial
    $ 354 "Serial Bridge uR0"
    SerialResponse = WTSerialBridge.send_command("/dev/ttyUSB0",1200, 8, "None", "One", "None", 1000, "None", "None", [252,82,48], False)
    # end: URCap Program Node
    $ 355 "Wait: 1.0"
    sleep(1.0)
    $ 356 "Set DO[0]=Off"
    set_standard_digital_out(0, False)
    $ 357 "'slice'"
    # 'slice'
    $ 358 "MoveL"
    $ 359 "Waypoint_21" "breakAfter"
    movel(Waypoint_21_p, a=0.05, v=0.03)
    $ 360 "Waypoint_42" "breakAfter"
    movel(Waypoint_42_p, a=0.05, v=0.03)
    $ 361 "Waypoint_43" "breakAfter"
    movel(Waypoint_43_p, a=0.05, v=0.03)
    $ 362 "Waypoint_44" "breakAfter"
    movel(Waypoint_44_p, a=0.05, v=0.03)
    $ 363 "Waypoint_74" "breakAfter"
    movel(Waypoint_74_p, a=0.05, v=0.03)
    $ 364 "MoveJ"
    $ 365 "Waypoint_45" "breakAfter"
    movej(get_inverse_kin(Waypoint_45_p, qnear=Waypoint_45_q), a=1.3962634015954636, v=1.0471975511965976)
    $ 366 "'above waypoint is home'"
    # 'above waypoint is home'
  end
  def align_tcp_forward():
    $ 368 "align_tcp_forward" "noBreak"
    $ 369 "'this program aligns the tcp parallel to the y direction'"
    # 'this program aligns the tcp parallel to the y direction'
    $ 370 "cp≔get_actual_tcp_pose()"
    global cp= get_actual_tcp_pose ()
    $ 371 "aligned_y_pose≔p[cp[0],cp[1],cp[2],0,-1.570796,0]"
    global aligned_y_pose=p[cp[0],cp[1],cp[2],0,-1.570796,0]
    $ 372 "MoveJ"
    $ 373 "aligned_y_pose" "breakAfter"
    movej(aligned_y_pose, a=1.3962634015954636, v=1.0471975511965976)
  end
  def align_tcp_up():
    $ 374 "align_tcp_up" "noBreak"
    $ 375 "'this program aligns the tcp parallel to the y direction'"
    # 'this program aligns the tcp parallel to the y direction'
    $ 376 "cp≔get_actual_tcp_pose()"
    global cp= get_actual_tcp_pose ()
    $ 377 "aligned_y_pose≔p[cp[0],cp[1],cp[2],0,0,0]"
    global aligned_y_pose=p[cp[0],cp[1],cp[2],0,0,0]
    $ 378 "MoveJ"
    $ 379 "aligned_y_pose" "breakAfter"
    movej(aligned_y_pose, a=1.3962634015954636, v=1.0471975511965976)
  end
  def align_ready_for_welding():
    $ 380 "align_ready_for_welding" "noBreak"
    $ 381 "'this program takes the welder from home to a position alined ready for welding (vertically down)'"
    # 'this program takes the welder from home to a position alined ready for welding (vertically down)'
    $ 382 "MoveJ"
    $ 383 "oldhome" "breakAfter"
    movej(get_inverse_kin(oldhome_p, qnear=oldhome_q), a=1.3962634015954636, v=1.0471975511965976)
    $ 384 "Waypoint_34" "breakAfter"
    movej(get_inverse_kin(Waypoint_34_p, qnear=Waypoint_34_q), a=1.3962634015954636, v=1.0471975511965976)
    $ 385 "Waypoint_35" "breakAfter"
    movej(get_inverse_kin(Waypoint_35_p, qnear=Waypoint_35_q), a=1.3962634015954636, v=1.0471975511965976)
    $ 386 "Waypoint_36" "breakAfter"
    movej(get_inverse_kin(Waypoint_36_p, qnear=Waypoint_36_q), a=1.3962634015954636, v=1.0471975511965976)
  end
  def Corner_Homing_45():
    $ 387 "Corner_Homing_45" "noBreak"
    $ 388 "'Use this program when tool is already positioned close to corner at 45deg'"
    # 'Use this program when tool is already positioned close to corner at 45deg'
    $ 389 "'tool flange will seek all 3 sides. will save those 5 locs in p__'"
    # 'tool flange will seek all 3 sides. will save those 5 locs in p__'
    $ 390 "Set"
    set_tcp(p[0.0,-0.004,0.284,0.0,0.0,0.0])
    $ 391 "'dummy move below for debug'"
    # 'dummy move below for debug'
    $ 396 "Wait: 1.0"
    sleep(1.0)
    $ 397 "tp≔get_actual_tcp_pose()"
    global tp= get_actual_tcp_pose ()
    $ 398 "Script: analyze_touchpoints.script"
    # this file creates the function for analyzing touchpoints
    # define pi
    pi = 3.1415926535

    # this is the main entry point for calculations.
    # it takes in the 5 points, analyzes the shape of the box, and then calculates path points and returns them
    # specifically for Down, Over, then Around (DOtA)
    # specifically for right-sided boxes (vertical weld on right side of edge)
    def main_calculate_right(p11, p12, p21, p22, p3, p13, p23):
        struct1 = analyze_touchpoints_only(p11, p12, p21, p22, p3)
        list1 = analyze_vertical_touchpoints(p11, p12, p13, p21, p22, p23, p3)
        struct2 = calculate_DOtA_points_right(struct1, list1)
        validity = check_validity_right(struct1, struct2)
        return struct2
    end

    # this is the main entry point for calculations.
    # it takes in the 5 points, analyzes the shape of the box, and then calculates path points and returns them
    # specifically for Down, Over, then Around (DOtA)
    # specifically for left-sided boxes (vertical weld on left side of edge)
    def main_calculate_left(p11, p12, p21, p22, p3, p13, p23):
        struct1 = analyze_touchpoints_only(p11, p12, p21, p22, p3)
        list1 = analyze_vertical_touchpoints(p11, p12, p13, p21, p22, p23, p3)
        struct2 = calculate_DOtA_points_left(struct1, list1)
        validity = check_validity_left(struct1, struct2)
        return struct2
    end

    # it takes 5 arguments as points
    # it returns a struct containing: (pointintersect, pointapproach1, pointapproach2, point1, point2, point3, point4, point5, pointreturn1, heading1, heading2, heading3, path2r1, path2r2, path2l1, path2l2)
    # specifically for Around then Up (AtU)
    def analyze_touchpoints(p11, p12, p21, p22, p3):
      # FIND THE INTERSECTION
      # comment get the z
      zcoord=p3[2]

      # get the raw points from the first line
      l1p1x=p11[0]
      l1p1y=p11[1]
      l1p2x=p12[0]
      l1p2y=p12[1]

      # equate the first line in 2d space
      ml1 = (l1p2y-l1p1y) / (l1p2x-l1p1x)

      # b = y - mx
      bl1 = l1p1y - ml1 * l1p1x

      # get the raw points from the second line
      l2p1x=p21[0]
      l2p1y=p21[1]
      l2p2x=p22[0]
      l2p2y=p22[1]

      # equate the second line in 2d space
      ml2 = (l2p2y-l2p1y) / (l2p2x-l2p1x)

      # b = y - mx
      bl2 = l2p1y - ml2 * l2p1x


      # find the intersection of the two lines
      # m1x+b1 = m2x+b2
      # m1x - m2x = b2 - b1
      # x = (b2-b1) / (m1-m2)
      xintersect = (bl2-bl1) / (ml1-ml2)
      yintersect = ml1 * xintersect + bl1

      #FIND THE VECTORS
      #define a vector from the intersection to the second point on the first line
      l1delxfull = l1p2x - xintersect
      l1delyfull = l1p2y - yintersect

      l1delmag = sqrt(l1delxfull*l1delxfull + l1delyfull*l1delyfull)

      l1delxunit = l1delxfull / l1delmag
      l1delyunit = l1delyfull / l1delmag

      #define a vector from the intersection to the second point on the second line
      l2delxfull = l2p2x - xintersect
      l2delyfull = l2p2y - yintersect

      l2delmag = sqrt(l2delxfull*l2delxfull + l2delyfull*l2delyfull)

      l2delxunit = l2delxfull / l2delmag
      l2delyunit = l2delyfull / l2delmag

      # FIND THE FOUR POINTS ON THE LINES
      # find locations 8 inches away from  intersect point
      # CONST
      welddistance = 8
      roundoverdistance = 0.05
      zup = .375
      # inches
      wd = welddistance * 25.4 / 1000
      rod = roundoverdistance * 25.4 / 1000
      zup = zup * 25.4 / 1000

      # now we have the unit vector. extend the weld distance from the intersection
      x = xintersect + l1delxunit * wd
      y = yintersect + l1delyunit * wd
      z = zcoord + zup

      point1 = p[x,y,z,1.570796,0,0] # dummy orientation for now

      x = xintersect + l1delxunit * rod
      y = yintersect + l1delyunit * rod

      point2 = p[x,y,z,1.570796,0,0]

      # now we have the unit vector. extend the weld distance from the intersection
      x = xintersect + l2delxunit * wd
      y = yintersect + l2delyunit * wd

      point5 = p[x,y,z,0,-1.570796,0]

      x = xintersect + l2delxunit * rod
      y = yintersect + l2delyunit * rod

      point4 = p[x,y,z,0,-1.570796,0]

      #DEFINE APPROACH POINTS
      pointintersect = p[xintersect,yintersect,zcoord,0,0,0]
      pointapproach1 = p[xintersect+0.1,yintersect+0.1,z,1.570796,0,0]
      pointapproach2 = p[point1[0], point1[1]+0.1, point1[2], point1[3], point1[4], point1[5]]
      pointreturn1 = p[point5[0]+0.1, point5[1], point5[2], point5[3], point5[4], point5[5]]

      #FIND HEADINGS
      #for each heading, find the angle of the line with respect to the pos x axis. then add/subtract 90 degrees because you want to be perpendicular to that
      headingvector1 = convert_uv_to_heading(l1delxunit, l1delyunit)
      headingvector2 = convert_uv_to_heading(l2delxunit, l2delyunit)
      # find halfway heading
      heading2 = (headingvector1 + headingvector2)/2
      # find headings that the robot should face while traveling, perpendicular to the vectors of the sides of the box
      heading1 = headingvector1 + pi/2
      heading3 = headingvector2 - pi/2

      #FIND POINT 3
      #see if we have to / can find point 3
      findpoint3 = True
      if roundoverdistance == 0:
        findpoint3 = False
      end
      if findpoint3:
        # i need to find the point3 such that the arc from p2 to p3 to p4 is tangent to p1-p2 and p4-p5. making this a smooth path will be good
        # the direction of movement is from pointintersect in the direction of heading2
        # how much movement though? this will depend on whether it is actually a 90 degree angle or not.
        # first, find the perpendicular lines through points 2 and 4
        perp2 = find_perpendicular_line(ml1, point2[0], point2[1])
        perp4 = find_perpendicular_line(ml2, point4[0], point4[1])
        # next, find the intersection of those two lines
        perpintersect = find_intersection(perp2[0], perp2[1], perp4[0], perp4[1])
        radiusofcircle = distance_between(perpintersect[0], perpintersect[1], 0, point2[0], point2[1], 0)
        # find a vector the direction of heading2
        uvx = cos(heading2)
        uvy = sin(heading2)
        # compute point3. pass in negative radius because the direction is into the tank but we want to move from the intersection out to the rounded edge.
        point3coords = add_vectordistance_to_point(perpintersect[0], perpintersect[1], z, uvx, uvy, 0, -1 * radiusofcircle)
        point3 = p[point3coords[0], point3coords[1], point3coords[2], 0, 0, 0]
      end

      #APPLY ACTUAL RXRYRZ TO POINTS
      # convert the headings to rxryrz and insert those values into the relevant points
      rxryrz = convert_heading_to_axang(heading1)
      rx = rxryrz[0]
      ry = rxryrz[1]
      rz = rxryrz[2]
      pointapproach1 = p[pointapproach1[0], pointapproach1[1], pointapproach1[2], rx, ry, rz]
      pointapproach2 = p[pointapproach2[0], pointapproach2[1], pointapproach2[2], rx, ry, rz]
      point1 = p[point1[0], point1[1], point1[2], rx, ry, rz]
      point2 = p[point2[0], point2[1], point2[2], rx, ry, rz]
      rxryrz = convert_heading_to_axang(heading2)
      rx = rxryrz[0]
      ry = rxryrz[1]
      rz = rxryrz[2]
      if findpoint3:
        point3 = p[point3[0], point3[1], point3[2], rx, ry, rz]
      else:
        point3 = point2
      end
      rxryrz = convert_heading_to_axang(heading3)
      rx = rxryrz[0]
      ry = rxryrz[1]
      rz = rxryrz[2]
      point4 = p[point4[0], point4[1], point4[2], rx, ry, rz]
      point5 = p[point5[0], point5[1], point5[2], rx, ry, rz]
      pointreturn1 = p[pointreturn1[0], pointreturn1[1], pointreturn1[2], rx, ry, rz]

      #find path2 (the part that goes up)
      four_vertical_points = find_vertical_points(pointintersect, l1delxunit, l1delyunit, l2delxunit, l2delyunit, zup, wd, heading1, heading3)
      path2r1 = four_vertical_points[0]
      path2r2 = four_vertical_points[1]
      path2l1 = four_vertical_points[2]
      path2l2 = four_vertical_points[3]

      #RETURN STRUCT
      ret = struct(pointintersect=pointintersect, pointapproach1=pointapproach1, pointapproach2=pointapproach2, point1=point1, point2=point2, point3=point3, point4=point4, point5=point5, pointreturn1=pointreturn1, heading1=heading1, heading2=heading2, heading3=heading3, path2r1=path2r1, path2r2=path2r2, path2l1=path2l1, path2l2=path2l2)
      return ret
    end

    # it takes 5 arguments as points
    # it returns a struct containing: (pointintersect, heading1, heading2, heading3, l1delxunit, l1delyunit, l2delxunit, l2delyunit)
    def analyze_touchpoints_only(p11, p12, p21, p22, p3):
      # FIND THE INTERSECTION
      # comment get the z
      zcoord=p3[2]

      # get the raw points from the first line
      l1p1x=p11[0]
      l1p1y=p11[1]
      l1p2x=p12[0]
      l1p2y=p12[1]

      # equate the first line in 2d space
      ml1 = (l1p2y-l1p1y) / (l1p2x-l1p1x)

      # b = y - mx
      bl1 = l1p1y - ml1 * l1p1x

      # get the raw points from the second line
      l2p1x=p21[0]
      l2p1y=p21[1]
      l2p2x=p22[0]
      l2p2y=p22[1]

      # equate the second line in 2d space
      ml2 = (l2p2y-l2p1y) / (l2p2x-l2p1x)

      # b = y - mx
      bl2 = l2p1y - ml2 * l2p1x


      # find the intersection of the two lines
      # m1x+b1 = m2x+b2
      # m1x - m2x = b2 - b1
      # x = (b2-b1) / (m1-m2)
      xintersect = (bl2-bl1) / (ml1-ml2)
      yintersect = ml1 * xintersect + bl1

      pointintersect = p[xintersect,yintersect,zcoord,0,0,0]

      #FIND THE VECTORS
      #define a vector from the intersection to the second point on the first line
      l1delxfull = l1p2x - xintersect
      l1delyfull = l1p2y - yintersect

      l1delmag = sqrt(l1delxfull*l1delxfull + l1delyfull*l1delyfull)

      l1delxunit = l1delxfull / l1delmag
      l1delyunit = l1delyfull / l1delmag

      #define a vector from the intersection to the second point on the second line
      l2delxfull = l2p2x - xintersect
      l2delyfull = l2p2y - yintersect

      l2delmag = sqrt(l2delxfull*l2delxfull + l2delyfull*l2delyfull)

      l2delxunit = l2delxfull / l2delmag
      l2delyunit = l2delyfull / l2delmag

      #FIND HEADINGS
      #for each heading, find the angle of the line with respect to the pos x axis. then add/subtract 90 degrees because you want to be perpendicular to that
      headingvector1 = convert_uv_to_heading(l1delxunit, l1delyunit)
      headingvector2 = convert_uv_to_heading(l2delxunit, l2delyunit)
      # find halfway heading
      heading2 = (headingvector1 + headingvector2)/2
      # find headings that the robot should face while traveling, perpendicular to the vectors of the sides of the box
      heading1 = headingvector1 + pi/2
      heading3 = headingvector2 - pi/2

      #RETURN STRUCT
      ret = struct(pointintersect=pointintersect, heading1=heading1, heading2=heading2, heading3=heading3, l1delxunit=l1delxunit, l1delyunit=l1delyunit, l2delxunit=l2delxunit, l2delyunit=l2delyunit)
      return ret
    end

    # given a struct from analyze_touchpoints_only(), calculate the points
    def calculate_DOtA_points_right(struct1, listleans):
        # get the stuff from the struct
        pointintersect = struct1[0]
        heading1 = struct1[1]
        heading2 = struct1[2]
        heading3 = struct1[3]
        l1delxunit = struct1[4]
        l1delyunit = struct1[5]
        l2delxunit = struct1[6]
        l2delyunit = struct1[7]

        # FIND THE POINTS ON THE LINES OF THE FIRST TURN PATH
        # find locations 8 inches away from  intersect point
        # CONST
        welddistance1 = 8 # vertical weld distance
        welddistance2 = 6 # first path second leg
        welddistance3 = 8 # second path second leg
        zup = .375
        # inches
        wd1 = welddistance1 * 25.4 / 1000
        wd2 = welddistance2 * 25.4 / 1000
        wd3 = welddistance3 * 25.4 / 1000
        zup = zup * 25.4 / 1000

        x = pointintersect[0] + l1delxunit * zup
        y = pointintersect[1] + l1delyunit * zup
        z = pointintersect[2] + zup

        #apply actual rxryrz to points
        # convert the headings to rxryrz and insert those values into the relevant points
        rxryrz = convert_heading_to_axang_preheatdown(heading1)
        rx = rxryrz[0]
        ry = rxryrz[1]
        rz = rxryrz[2]

        point1 = p[x + wd1*listleans[0], y + wd1*listleans[1], z + wd1, rx, ry, rz] # add in the listleans factor to follow the face of the box as we move up
        point2 = p[x, y, z, rx, ry, rz]

        # convert the headings to rxryrz and insert those values into the relevant points
        rxryrz = convert_heading_to_axang_ccw(heading1)
        rx = rxryrz[0]
        ry = rxryrz[1]
        rz = rxryrz[2]

        point4 = p[x, y, z, rx, ry, rz]
        x = x + l1delxunit * wd2
        y = y + l1delyunit * wd2
        point5 = p[x, y, z, rx, ry, rz]

        # FIND THE POINTS ON THE LINES OF THE SECOND AROUND PATH
        roundoverdistance = 0.05
        rod = roundoverdistance * 25.4 / 1000

        # now we have the unit vector. extend the weld distance from the intersection
        x = pointintersect[0] + l1delxunit * (zup)
        y = pointintersect[1] + l1delyunit * zup
        # convert the headings to rxryrz and insert those values into the relevant points
        rxryrz = convert_heading_to_axang(heading1)
        rx = rxryrz[0]
        ry = rxryrz[1]
        rz = rxryrz[2]
        point_1 = p[x, y, z, rx, ry, rz]

        x = pointintersect[0] + l1delxunit * rod
        y = pointintersect[1] + l1delyunit * rod
        point_2 = p[x, y, z, rx, ry, rz]

        # now we have the unit vector. extend the weld distance from the intersection
        x = pointintersect[0] + l2delxunit * wd3
        y = pointintersect[1] + l2delyunit * wd3
        # convert the headings to rxryrz and insert those values into the relevant points
        rxryrz = convert_heading_to_axang(heading3)
        rx = rxryrz[0]
        ry = rxryrz[1]
        rz = rxryrz[2]
        point_5 = p[x, y, z, rx, ry, rz]

        x = pointintersect[0] + l2delxunit * rod
        y = pointintersect[1] + l2delyunit * rod
        point_4 = p[x, y, z, rx, ry, rz]

        #FIND POINT 3
        # by calling analyze_touchpoints()
        atret = analyze_touchpoints(point_2, point_1, point_4, point_5, pointintersect)
        point_3 = atret[5]


        struct2 = struct(point1=point1, point2=point2, point4=point4, point5=point5, point_1=point_1, point_2=point_2, point_3=point_3, point_4=point_4, point_5=point_5)
        return struct2
    end

    # given a struct from analyze_touchpoints_only(), calculate the points
    def calculate_DOtA_points_left(struct1, listleans):
        # get the stuff from the struct
        pointintersect = struct1[0]
        heading1 = struct1[1]
        heading2 = struct1[2]
        heading3 = struct1[3]
        l1delxunit = struct1[4]
        l1delyunit = struct1[5]
        l2delxunit = struct1[6]
        l2delyunit = struct1[7]

        # FIND THE POINTS ON THE LINES OF THE FIRST TURN PATH
        # find locations 8 inches away from  intersect point
        # CONST
        welddistance1 = 8 # vertical weld distance
        welddistance2 = 6 # first path second leg
        welddistance3 = 8 # second path second leg
        zup = .375
        # inches
        wd1 = welddistance1 * 25.4 / 1000
        wd2 = welddistance2 * 25.4 / 1000
        wd3 = welddistance3 * 25.4 / 1000
        zup = zup * 25.4 / 1000

        x = pointintersect[0] + l2delxunit * zup
        y = pointintersect[1] + l2delyunit * zup
        z = pointintersect[2] + zup

        #apply actual rxryrz to points
        # convert the headings to rxryrz and insert those values into the relevant points
        rxryrz = convert_heading_to_axang_preheatdown(heading3)
        rx = rxryrz[0]
        ry = rxryrz[1]
        rz = rxryrz[2]

        point1 = p[x + wd1*listleans[0], y + wd1*listleans[1], z + wd1, rx, ry, rz]
        point2 = p[x, y, z, rx, ry, rz]

        # convert the headings to rxryrz and insert those values into the relevant points
        rxryrz = convert_heading_to_axang(heading3)
        rx = rxryrz[0]
        ry = rxryrz[1]
        rz = rxryrz[2]

        point4 = p[x, y, z, rx, ry, rz]
        x = x + l2delxunit * wd2
        y = y + l2delyunit * wd2
        point5 = p[x, y, z, rx, ry, rz]

        # FIND THE POINTS ON THE LINES OF THE SECOND AROUND PATH
        roundoverdistance = 0.05
        rod = roundoverdistance * 25.4 / 1000

        # now we have the unit vector. extend the weld distance from the intersection
        x = pointintersect[0] + l2delxunit * (zup)
        y = pointintersect[1] + l2delyunit * zup
        # convert the headings to rxryrz and insert those values into the relevant points
        rxryrz = convert_heading_to_axang_ccw(heading3)
        rx = rxryrz[0]
        ry = rxryrz[1]
        rz = rxryrz[2]
        point_1 = p[x, y, z, rx, ry, rz]

        x = pointintersect[0] + l2delxunit * rod
        y = pointintersect[1] + l2delyunit * rod
        point_2 = p[x, y, z, rx, ry, rz]

        # now we have the unit vector. extend the weld distance from the intersection
        x = pointintersect[0] + l1delxunit * wd3
        y = pointintersect[1] + l1delyunit * wd3
        # convert the headings to rxryrz and insert those values into the relevant points
        rxryrz = convert_heading_to_axang_ccw(heading1)
        rx = rxryrz[0]
        ry = rxryrz[1]
        rz = rxryrz[2]
        point_5 = p[x, y, z, rx, ry, rz]

        x = pointintersect[0] + l1delxunit * rod
        y = pointintersect[1] + l1delyunit * rod
        point_4 = p[x, y, z, rx, ry, rz]

        #FIND POINT 3
        # by calling analyze_touchpoints()
        atret = analyze_touchpoints(point_2, point_1, point_4, point_5, pointintersect)
        point_3 = atret[5]
        #point 3 will not have the correct rxryrz though because now the gun needs to be face up.
        rxryrz = convert_heading_to_axang_ccw(heading2)
        rx = rxryrz[0]
        ry = rxryrz[1]
        rz = rxryrz[2]
        point_3 = p[point_3[0], point_3[1], point_3[2], rx, ry, rz]

        struct2 = struct(point1=point1, point2=point2, point4=point4, point5=point5, point_1=point_1, point_2=point_2, point_3=point_3, point_4=point_4, point_5=point_5)
        return struct2
    end

    # this function analyzes the vertical points
    # calculates the slope of the edge in question
    # specifically, for each inch up in the z direction, what is the change in x and change in y direction
    # returns a list of [nx, ny]
    def analyze_vertical_touchpoints(p11, p12, p13, p21, p22, p23, p3):
        # first, find the equations of the planes from the 6 points
        plane1 = findplane(p11, p12, p13)
        plane2 = findplane(p21, p22, p23)
        # Find the Direction Vector of the Line: The direction vector d of the line of intersection can be found by taking the cross product of the normal vectors of each plane (a, b, and c)
        nx = plane1[1]*plane2[2] - plane1[2]*plane2[1]
        ny = plane1[2]*plane2[0] - plane1[0]*plane2[2]
        nz = plane1[0]*plane2[1] - plane1[1]*plane2[0]
        # normalize the vector so the z length is 1
        multiplier = 1 / nz
        nx = nx * multiplier
        ny = ny * multiplier
        nz = nz * multiplier # should become equal to 1
        ret = [nx, ny]
        return ret
    end

    # given 3 points, this finds the plane and its equation
    # rereturns ax + by + cz + d = 0 in a list of [a, b, c, d]
    def findplane(p11, p12, p13):
        # extract coordinates
        x1 = p11[0]
        y1 = p11[1]
        z1 = p11[2]
        x2 = p12[0]
        y2 = p12[1]
        z2 = p12[2]
        x3 = p13[0]
        y3 = p13[1]
        z3 = p13[2]
        # create vectors from the points
        v1x = x2-x1
        v1y = y2-y1
        v1z = z2-z1
        v2x = x3-x1
        v2y = y3-y1
        v2z = z3-z1
        #calculate the normal vector using the cross product
        nx = v1y*v2z - v1z*v2y # i component
        ny = v1z*v2x - v1x*v2z # j component
        nz = v1x*v2y - v1y*v2x # k component
        # calculate d in the plane equation
        d = -1 * (nx*x1 + ny*y1 + nz*z1)
        ret = [nx, ny, nz, d]
        return ret
    end

    # given a heading, (ccw from +x axis), find the mx+b slope
    # fails if exactly vertical
    def get_slope_from_heading(heading):
        return tan(heading)
    end



    # this function finds the points (and rxryrz) of the 2 points (start and end) of vertical weld section
    def find_vertical_points(pointintersect, l1delxunit, l1delyunit, l2delxunit, l2delyunit, offset, wd, heading1, heading3):

      # find right side stuff
      # find the point in 3d space that is .375 up and .375 over
      x = pointintersect[0] + l1delxunit * offset
      y = pointintersect[1] + l1delyunit * offset
      z = pointintersect[2] + offset
      # find rxryrz
      rxryrz = convert_heading_to_axang_preheatup(heading1)
      rx = rxryrz[0]
      ry = rxryrz[1]
      rz = rxryrz[2]
      path2r1 = p[x, y, z, rx, ry, rz]
      path2r2 = p[x, y, z + wd, rx, ry, rz]

      # find left side
      # find the point in 3d space that is .375 up and .375 over
      x = pointintersect[0] + l2delxunit * offset
      y = pointintersect[1] + l2delyunit * offset
      z = pointintersect[2] + offset
      # find rxryrz
      rxryrz = convert_heading_to_axang_preheatup(heading3)
      rx = rxryrz[0]
      ry = rxryrz[1]
      rz = rxryrz[2]
      path2l1 = p[x, y, z, rx, ry, rz]
      path2l2 = p[x, y, z + wd, rx, ry, rz]

      ret = struct(path2r1=path2r1, path2r2=path2r2, path2l1=path2l1, path2l2=path2l2)
      return ret
    end

    # this function converts a unit vector to its heading angle ccw from x+ axis
    # takes uvx and uvy
    # returns heading in radians
    def convert_uv_to_heading(uvx, uvy):
      baseang = atan(uvy/uvx)
      if uvx < 0:
        ang = baseang + pi
      elif uvy < 0:
        ang = baseang + pi * 2
      else:
        ang = baseang
      end
      return ang
    end

    # this function finds the equation of a line, perpendicular to a given line, and going through a given point
    # takes 3 arguments: m (the original line's slope), x (point's x coord), y (point's y coord). the b of the original line is not needed
    # returns a list of [m,b] (the slope and intercept of the new line)
    def find_perpendicular_line(origm, x, y):
      m = (1/origm) * -1
      b = y - m*x
      ret = [m, b]
      return ret
    end

    # this function finds the intersection point between two lines in the xy plane
    # takes 4 arguments: m1, b1, m2, b2
    # returns a list of [x,y] (the point of intersection)
    def find_intersection(m1, b1, m2, b2):
      # m1x+b1 = m2x+b2
      # m1x - m2x = b2 - b1
      # x = (b2-b1) / (m1-m2)
      x = (b2-b1) / (m1-m2)
      y = m1 * x + b1
      ret = [x, y]
      return ret
    end

    # this function finds the distance between 2 points in 3d space
    # it takes 6 arguments: x1, y1, z1, x2, y2, z2
    # it returns a distance
    def distance_between(x1, y1, z1, x2, y2, z2):
      distsquared = (x2-x1)*(x2-x1)+(y2-y1)*(y2-y1)+(z2-z1)*(z2-z1)
      dist = sqrt(distsquared)
      return dist
    end

    # this function takes a point, a unit vector, and a distance, and adds the distance to the point in the direction of the unit vector (3d space)
    # it returns a point as a list of coordinates
    def add_vectordistance_to_point(xi, yi, zi, uvx, uvy, uvz, delta):
      xf = xi + uvx * delta
      yf = yi + uvy * delta
      zf = zi + uvz * delta
      ret = [xf, yf, zf]
      return ret
    end

    # this function converts a heading (ccw radians from the positive x axis) into rxryrz to be put into a point p[]
    # this will point the gun in this heading with the bottom side of the gun facing up.
    # the values used in this program were calculated by doing rotation matrix math in the file on WI-CALVINB10 C. Documents. Theory for converting rotations into axis angle representations
    def convert_heading_to_axang(heading):
     axisxraw = -1 * sin(heading)
     axisyraw = cos(heading) + 1
     axiszraw = sin(heading)

     magnitude = sqrt(axisxraw*axisxraw + axisyraw*axisyraw + axiszraw*axiszraw)

     axisxunit = axisxraw / magnitude
     axisyunit = axisyraw / magnitude
     axiszunit = axiszraw / magnitude

     angle = acos( (cos(heading) - 1) / 2 )

     rxout = axisxunit * angle
     ryout = axisyunit * angle
     rzout = axiszunit * angle

     return [rxout, ryout, rzout]
    end

    # this function converts a heading (ccw radians from the positive x axis) into rxryrz to be put into a point p[]
    # this will point the gun in this heading with the preheat side of the gun tip facing up. Used for welding in a vertical path.
    # the values used in this program were calculated by doing rotation matrix math in the file on WI-CALVINB10 C. Documents. Theory for converting rotations into axis angle representations
    def convert_heading_to_axang_preheatup(heading):
     axisxraw = -sin(heading) + 1
     axisyraw = cos(heading)
     axiszraw = cos(heading)

     magnitude = sqrt(axisxraw*axisxraw + axisyraw*axisyraw + axiszraw*axiszraw)

     axisxunit = axisxraw / magnitude
     axisyunit = axisyraw / magnitude
     axiszunit = axiszraw / magnitude

     angle = acos( (-sin(heading) - 1) / 2 )

     rxout = axisxunit * angle
     ryout = axisyunit * angle
     rzout = axiszunit * angle

     return [rxout, ryout, rzout]
    end

    # this function converts a heading (ccw radians from the positive x axis) into rxryrz to be put into a point p[]
    # this will point the gun in this heading with the preheat side of the gun tip facing down. Used for welding in a vertical path downwards.
    # the values used in this program were calculated by doing rotation matrix math in the file on WI-CALVINB10 C. Documents. Theory for converting rotations into axis angle representations
    def convert_heading_to_axang_preheatdown(heading):
     axisxraw = -sin(heading) - 1
     axisyraw = cos(heading)
     axiszraw = -cos(heading)

     magnitude = sqrt(axisxraw*axisxraw + axisyraw*axisyraw + axiszraw*axiszraw)

     axisxunit = axisxraw / magnitude
     axisyunit = axisyraw / magnitude
     axiszunit = axiszraw / magnitude

     angle = acos( (sin(heading) - 1) / 2 )

     rxout = axisxunit * angle
     ryout = axisyunit * angle
     rzout = axiszunit * angle

     return [rxout, ryout, rzout]
    end

    # this function converts a heading (ccw radians from the positive x axis) into rxryrz to be put into a point p[]
    # this will point the gun in this heading with the preheat side of the gun tip facing right. Used for welding counterclockwise around the box.
    # the values used in this program were calculated by doing rotation matrix math in the file on WI-CALVINB10 C. Documents. Theory for converting rotations into axis angle representations
    def convert_heading_to_axang_ccw(heading):
     axisxraw = -sin(heading)
     axisyraw = cos(heading) - 1
     axiszraw = -sin(heading)

     magnitude = sqrt(axisxraw*axisxraw + axisyraw*axisyraw + axiszraw*axiszraw)

     axisxunit = axisxraw / magnitude
     axisyunit = axisyraw / magnitude
     axiszunit = axiszraw / magnitude

     angle = acos( (-cos(heading) - 1) / 2 )

     rxout = axisxunit * angle
     ryout = axisyunit * angle
     rzout = axiszunit * angle

     return [rxout, ryout, rzout]
    end

    # this function is for getting the points along the path of the corner homing 45
    # point0 is the point where they touched
    def get_corner_homing_45_pathpoints(point0):
      p0x = point0[0]
      p0y = point0[1]
      p0z = point0[2]
      p0rx = point0[3]
      p0ry = point0[4]
      p0rz = point0[5]

      #constants
      #distances of how far away from point the touchpoints are
      d0 = 0.10 # how far from the box to retreat and approach
      d1 = 0.03 # first distance from init point
      d2 = 0.15 # second distance from init point
      d3 = 0.125 #vertical distance from first point
      sqrt2 = 0.707106781 # 1/sqrt(2) , the inverse of the sqrt(2)

      ph1 = p[p0x + d0, p0y, p0z + d1, p0rx, p0ry, p0rz] #approach point for turn

      ph2 = p[p0x+d0-d0*0.5-sqrt2*d1, p0y+d0*0.5+sqrt2*d1, p0z+d1, 1.446, -0.8, -0.733]
      ph3 = p[p0x+d0-d0*0.5-sqrt2*d2, p0y+d0*0.5+sqrt2*d2, p0z+d1, 1.446, -0.8, -0.733]
      ph4 = p[p0x+d0-d0*0.5-sqrt2*d1, p0y-d0*0.5-sqrt2*d1, p0z+d1, 0.626, -1.993, -1.813]
      ph5 = p[p0x+d0-d0*0.5-sqrt2*d2, p0y-d0*0.5-sqrt2*d2, p0z+d1, 0.626, -1.993, -1.813]

      # go back to ph1
      ph6 = p[p0x + d0, p0y, p0z -0.05, 0, 0, 0] # approach point for under turn
      # moveL from ph1 to ph6
      ph7 = p[p0x-d1, p0y, p0z-0.05, 0, 0, 0]

      # add the vertical touch points
      ph2up = p[ph2[0], ph2[1], ph2[2]+d3, ph2[3], ph2[4], ph2[5]]
      ph4up = p[ph4[0], ph4[1], ph4[2]+d3, ph4[3], ph4[4], ph4[5]]
      ret = struct(ph1=ph1, ph2=ph2, ph3=ph3, ph4=ph4, ph5=ph5, ph6=ph6, ph7=ph7, ph2up=ph2up, ph4up=ph4up)
      is_robot_at_reachable_spot(point0, ret)
      return ret
    end

    # this function checks whether the touchpoints are reachable AKA is the robot positioned in the right spot
    # if everything looks good, it continues.
    # if it detects a problem, it infinite loops a popup
    def is_robot_at_reachable_spot(point0, struct_touchpoints):
      # first, check whether the corner is too low to the ground that the bottom homing will hit the ground (z < -350)
      if point0[2] < -0.350:
        # bad
        popuptext = "Tank Corner is too low to the ground. Collisions will occur. Stop Program and raise tank. "
        # infinite loop
        while 1==1:
          popup(popuptext, title="Robot Positioning Warning",blocking=True)
        end
      end



      # next, check whether the touchpoints are reachable
      structlength = 9
      i = 0
      allvalid = True
      listproblems = ""
      listnames = ["ph1", "ph2", "ph3", "ph4", "ph5", "ph6", "ph7", "ph2up", "ph4up"]
      while i < structlength:
        curr = struct_touchpoints[i]
        valid = get_inverse_kin_has_solution(curr)
        if not valid:
          allvalid = False
          listproblems = listproblems + listnames[i]
        end
        i = i + 1
      end

      if not allvalid:
        # display
        popuptext = "Robot is too far from tank corner. Cannot reach some necessary positions. Stop Program and move robot closer. " + listproblems
        # infinite loop
        while 1==1:
          popup(popuptext, title="Robot Positioning Warning",blocking=True)
        end
      end

    end

    # checks the validity of all points during a left weld
    def check_validity_left(struct1, struct2):
      #first, check whether robot is too close
      pointintersect = struct1[0]
      # next, check if the corner is too close to the robot to do a left around weld (complex but approximately X > -1300)
      # if y < 0, then x < -1300. if y < 480, then y > (1300+x)*8. if y > 480, then y > (1235+x)*4 + 500
      toocloseleftweld = False
      if pointintersect[1] < 0:
        if pointintersect[0] > -1.300:
          toocloseleftweld = True
        end
      elif pointintersect[1] < 0.480:
        if pointintersect[1] < (1.300 + pointintersect[0])*8:
          toocloseleftweld = True
        end
      else:
        if pointintersect[1] < (1.235 + pointintersect[0])*4 + 0.500:
          toocloseleftweld = True
        end
      end
      if toocloseleftweld:
        # bad
        popuptext = "Robot is too close to tank corner. Collisions may occur. Stop Program and move robot farther. "
        # infinite loop
        while 1==1:
          popup(popuptext, title="Robot Positioning Warning",blocking=True)
        end
      end

      #next, check whether all the points in the weldpath are valid
      structlength = 9
      i = 0
      allvalid = True
      listproblems = ""
      listnames = ["point1", "point2", "point4", "point5", "point_1", "point_2", "point_3", "point_4", "point_5"]
      while i < structlength:
        curr = struct2[i]
        valid = get_inverse_kin_has_solution(curr)
        if not valid:
          allvalid = False
          listproblems = listproblems + listnames[i]
        end
        i = i + 1
      end

      if not allvalid:
        # display
        popuptext = "Robot is too far from tank corner. Cannot reach some necessary positions. Stop Program and move robot closer. " + listproblems
        # infinite loop
        while 1==1:
          popup(popuptext, title="Robot Positioning Warning",blocking=True)
        end
      end


    end

    # checks the validity of all points during a right weld
    def check_validity_right(struct1, struct2):
      # first, check whether the right pivot will bonk itself
      pointintersect = struct1[0]
      heading1 = struct1[1] # this is the direction that the welder will face when doing the right side of the box

      #first, check whether the heading is just too far offset
      # more than 15 degrees off of 45 is too much
      # normal heading is 216 degrees
      #201 degrees to 231 degrees
      heading1degrees = heading1 * 180 / pi
      if heading1degrees < 201 or heading1degrees > 231 :
        # then out of range
        popuptext = "Robot is not aligned at a 45 degree angle of corner (15 degree leeway). Collisions may occur. Stop Program and align robot. heading1degrees=" + str_cat("",heading1degrees)
        # infinite loop
        while 1==1:
          popup(popuptext, title="Robot Positioning Warning",blocking=True)
        end
      end

      #TODO: add the checks for whether x is too close, given the heading
      # add checks for whether x is too close, given the heading
      # different equations for whether heading offset > 5 degrees or less (inc. negative)
      headingoffset = heading1degrees - 216
      if headingoffset < 5:
        # then calculate a and b
        a = 0.4584 + -0.02369 * headingoffset
        b = (-1151.4 + 13.83 * headingoffset) / 1000
        # check whether x > a*y+b
        if pointintersect[0] > a * pointintersect[1] + b:
          # bad
          popuptext = "Robot is too close to tank corner or not at the right angle. Collisions may occur. Stop Program and align robot. "
          # infinite loop
          while 1==1:
            popup(popuptext, title="Robot Positioning Warning",blocking=True)
          end
        end
      else:
        # headingoffset > 5 degrees
        if pointintersect[1] < 0:
          if pointintersect[0] > -1150.0 / 1000.0:
            #bad
            popuptext = "Robot is too close to tank corner. Collisions may occur. Stop Program and align robot. "
            # infinite loop
            while 1==1:
              popup(popuptext, title="Robot Positioning Warning",blocking=True)
            end
          end
        else:
          # if x > .7736 y - 1101.9 then bad
          if pointintersect[0] > 0.7736 * pointintersect[1] - 1101.9 / 1000:
            popuptext = "Robot is too close to tank corner. Collisions may occur. Stop Program and align robot. "
            # infinite loop
            while 1==1:
              popup(popuptext, title="Robot Positioning Warning",blocking=True)
            end
          end
        end
      end

      #next, check whether all the points in the weldpath are valid
      structlength = 9
      i = 0
      allvalid = True
      listproblems = ""
      listnames = ["point1", "point2", "point4", "point5", "point_1", "point_2", "point_3", "point_4", "point_5"]
      while i < structlength:
        curr = struct2[i]
        valid = get_inverse_kin_has_solution(curr)
        if not valid:
          allvalid = False
          listproblems = listproblems + listnames[i]
        end
        i = i + 1
      end

      if not allvalid:
        # display
        popuptext = "Robot is too far from tank corner. Cannot reach some necessary positions. Stop Program and move robot closer. " + listproblems
        # infinite loop
        while 1==1:
          popup(popuptext, title="Robot Positioning Warning",blocking=True)
        end
      end
    end

    # this function sends a signal to turn extrusion on
    def turn_extrusion_on():
      # flush the channel
      resp0 = send_serial_signal(["u", "r", "?"])
      # send the signal
      resp1 = send_serial_signal(["u", "R", "1"])
      # if resp <> "uR1"
      if resp1 != [252,82,49]:
        # turn off extrusion and heating. inform calvin
        resp2 = send_serial_signal(["u", "R", "0"])
        resp3 = send_serial_signal(["u", "H", "0"])
        popuptext = "Error code encountered while trying to start extrusion. Find Calvin. "
        while 1==1:
          popup(popuptext, title="Extrusion Error Code",blocking=True)
          popup(resp1, blocking=True)
        end
      end
    end

    # this function sends a signal and receives a response
    # signal is a list of 3 strings, 1 character each. first is u. second is the next character. third is final character
    def send_serial_signal(signal):
      signal2char = signal[1]
      signal3char = signal[2]
      listsignal = [252, get_corr_number(signal2char), get_corr_number(signal3char)]
      resp1 = WTSerialBridge.send_command("/dev/ttyUSB0",1200, 8, "None", "One", "None", 1000, "None", "None", listsignal, True)
      return resp1
    end

    # this function converts a letter into its ascii number
    def get_corr_number(letter):
      if letter == "A":
        return 65
      elif letter == "H":
        return 72
      elif letter == "R":
        return 82
      elif letter == "M":
        return 77
      elif letter == "E":
        return 69
      elif letter == "a":
        return 97
      elif letter == "b":
        return 98
      elif letter == "h":
        return 104
      elif letter == "r":
        return 114
      elif letter == "s":
        return 115
      elif letter == "m":
        return 109
      elif letter == "0":
        return 48
      elif letter == "1":
        return 49
      elif letter == "2":
        return 50
      elif letter == "3":
        return 51
      elif letter == "4":
        return 52
      elif letter == "5":
        return 53
      elif letter == "6":
        return 54
      elif letter == "7":
        return 55
      elif letter == "8":
        return 56
      elif letter == "9":
        return 57
      elif letter == "?":
        return 63
      end
    end

    # this function checks whether the welder is in the ready state.
    # to be called at the beginning of Main Program
    def welder_state_ready():
      # flush the channel
      resp0 = send_serial_signal(["u", "s", "?"])
      # send the signal
      resp1 = send_serial_signal(["u", "s", "?"])
      # if resp1 == [252,115,49] (us1) then it is ready. otherwise, it is not
      if resp1 != [252,115,49]:
        popuptext = "Welder is not ready for extrusion. Follow the instructions to start heating welder. "
        while 1==1:
          popup(popuptext, title="Welder Not Ready",blocking=True)
        end
      end

